Universal Robots PolyScope program: GlueCeiling.urp

Program GlueCeiling (createdIn=3.0.0 lastSavedIn=3.0.0 directory=/programs installation=default)
Robot Program (runOnlyOnce=true motionType=MoveJ speed=1.047198 acceleration=1.396263 useActiveTCP=false)
  'Program generated by RoboDK v5.3.2 for UR5e on 20/01/2022 14:10:44'
  'Using nominal kinematics.'
  'Using Ref. Baia 1: p[0.136922, -0.316489, 0.045000, 0.000000, 0.000000, -0.785398]'
  Call approach_t1
  Call to1
  Call GluePath
  Call approach_t1
SubProgram -> approach_t1
SubProgram -> to1
SubProgram -> GluePath
SubProgram -> approach_t1
SubProgram -> to1
SubProgram -> GluePath
SubProgram -> approach_t1
SubProgram approach_t1 (keepSynchronizedWithDisk=true trackProgramExecution=false) programFile=/programs/approach_t1.urp
SubProgram to1 (keepSynchronizedWithDisk=true trackProgramExecution=false) programFile=/programs/to1.urp
SubProgram GluePath (keepSynchronizedWithDisk=true trackProgramExecution=false) programFile=/programs/GluePath.urp
